(*********************************** G.D S.p.A. - Technical Department ***********************************
============= PROGRAM INFO ============
FOLDER:             TBD
MACHINES INVOLVED:  TBD 

============= DESCRIPTION =============
csp machine declaration

============= REVISIONS ===============
Date		Version	 	Author      	Description             
----------	-------		------------  	--------------------------------------------
2019/04/05 	0000.00	 	M.Grasso		Creation of the PRG

**********************************************************************************************************)
(*$R process_ref := prc; $*)
PROGRAM csp_case_feed_magazine_accU
VAR
		
	prc:											process;
	prc_path:										STRING;
	
	
END_VAR

_read_var_input();

_object_manager();

IF NOT objects_running()
THEN
	RETURN;	
END_IF

_read_process_image();

_mode_manager();

_set_runtime_properties();

(********************************* BODY *********************************)


(************************************************************************)

_handle_messages();

_write_output();

ACTION _handle_messages:
;
END_ACTION

ACTION _handle_process_test:
;
END_ACTION

ACTION _mode_manager:
IF process_mode_req_is_pending(prc)
THEN
    process_apply_mode_req_first_step(prc);
    CASE process_get_mode(prc) OF
        MODE_TO_ABSENT:
			;
        MODE_TO_INACTIVE:
			;
        MODE_TO_TEST:
			;
        MODE_TO_OPERATIONAL:
			;
    END_CASE
    process_apply_mode_req_second_step(prc);
END_IF
END_ACTION

ACTION _object_manager:
IF objects_initialization()
THEN
	sub_process_init(
		object_name					:= 'csp_case_feed_magazine_accU.prc', 
		process						:= csp_case_feed_magazine.prc, 
		CONVERSION_this				:= prc);
		
	prc_path 						:= process_get_path(prc);
	
END_IF

IF objects_running()
THEN
	process_cycle(prc);
	
END_IF
END_ACTION

ACTION _read_process_image:
;
END_ACTION

ACTION _read_var_input:
;
END_ACTION

ACTION _set_runtime_properties:
;
END_ACTION

ACTION _write_output:
;
END_ACTION

END_PROGRAM

(* stored: Version 1.1.0.1, ProductVersion 3.1.4024.3
   POU csp_case_feed_magazine_accU: Id {d5fed557-2e0d-48bb-a72e-4f4c46c1ee12}, SpecialFunc None
   Action _handle_messages: Id {b139f7cf-acb6-47d4-b00d-f6e1e67822ba}
   Action _handle_process_test: Id {ec002bf9-18b3-41f1-9a38-4c7e02b21469}
   Action _mode_manager: Id {fb7eed95-16a0-447b-b76d-5534b152b250}
   Action _object_manager: Id {564cf3c8-b0ca-44f4-a4a6-b6ad86d0a9d9}
   Action _read_process_image: Id {cadbec6b-4fd2-46d9-b99f-13fc4a49d72d}
   Action _read_var_input: Id {7ef92c70-5a97-4ad9-8e70-de03610d4127}
   Action _set_runtime_properties: Id {13aa6d27-a470-4f85-a0ca-ec48af685ab9}
   Action _write_output: Id {55616371-abc6-4b15-b815-9dda8a82bbb3} *)
